(* CODESYS project ESSE.project

Project tree, tasks and I/O mapping:
  Device : CODESYS Control Win V3, 3S - Smart Software Solutions GmbH, order no. 305021, version 3.5.11.30
    application Application
      libraries: Standard, * (System)
      task MainTask (cyclic, interval t#20ms, priority 1) calls PLC_PRG
      program PLC_PRG [LD]
*)

// Device/Application/PLC_PRG
PROGRAM PLC_PRG
VAR
	B1 : BOOL;        // BOTAO 1  
    B2 : BOOL;        // BOTAO 2
	M1 : BOOL;        // MOTOR 1
	M2 : BOOL;        // MOTOR 2
	S1 : BOOL;        // sensor de peça
	S2 : BOOL;        // cortina de segurança
	S3 : BOOL;        // sensor de fim de curso 3
    S4 : BOOL;        // sensor de fim de curso 4
	L1 : BOOL;        // SISTEMA EM FUNCIONAMENTO
	L2 : BOOL;        // SISTEMA PARADO
	BE : BOOL;        // é um botão de emergência
	P1: BOOL;         // PASSO 1
	P3: BOOL;         // PASSO 3
	P2: BOOL;         // PASSO 2
	P4: BOOL;         // PASSO 4
	P5: BOOL;         // PASSO 5
	P6: BOOL;         // PASSO 6
END_VAR
VAR // added by the converter: edge detectors and wires of the graphical bodies
    _w1, _w2 : BOOL;
END_VAR

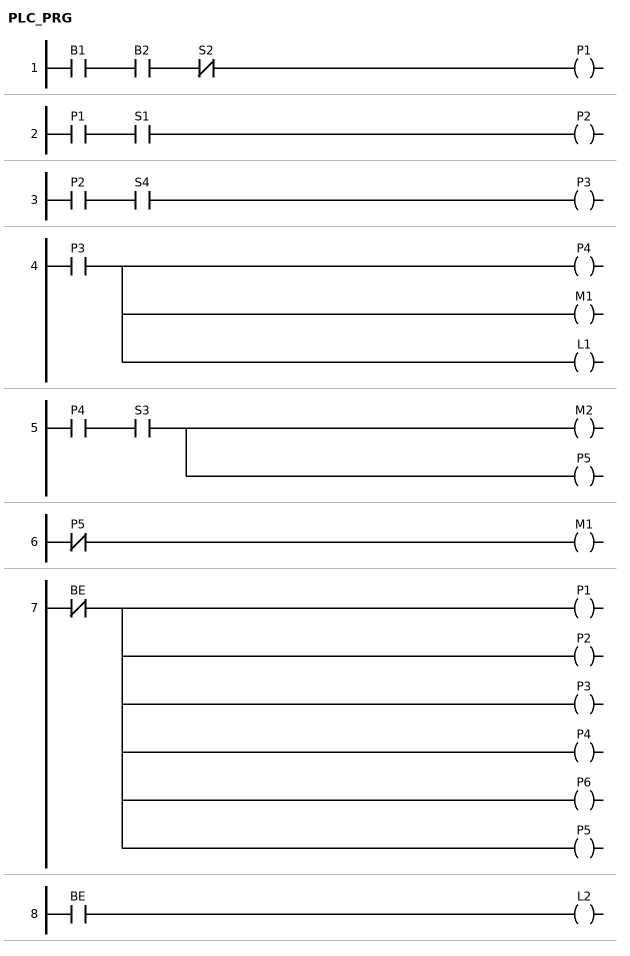
// NETWORK 1
P1 := B1 AND B2 AND NOT S2;

// NETWORK 2
P2 := P1 AND S1;

// NETWORK 3
P3 := P2 AND S4;

// NETWORK 4
P4 := P3;
M1 := P3;
L1 := P3;

// NETWORK 5
_w1 := P4 AND S3;
M2 := _w1;
P5 := _w1;

// NETWORK 6
M1 := NOT P5;

// NETWORK 7
_w2 := NOT BE;
P1 := _w2;
P2 := _w2;
P3 := _w2;
P4 := _w2;
P6 := _w2;
P5 := _w2;

// NETWORK 8
L2 := BE;

END_PROGRAM
